// TwinCAT 3 PLC project PLC_SJ_MOCVD
// ProgramVersion: 3.1.4023.0
// libraries:
//   Tc2_ControllerToolbox, * (Beckhoff Automation GmbH)
//   Tc2_IoFunctions, * (Beckhoff Automation GmbH)
//   Tc2_ModbusRTU, * (Beckhoff Automation GmbH)
//   Tc2_ModbusSrv, * (Beckhoff Automation GmbH)
//   Tc2_SerialCom, * (Beckhoff Automation GmbH)
//   Tc2_Standard, * (Beckhoff Automation GmbH)
//   Tc2_System, * (Beckhoff Automation GmbH)
//   Tc2_TempController, * (Beckhoff Automation GmbH)
//   Tc2_Utilities, * (Beckhoff Automation GmbH)
//   Tc3_Module, * (Beckhoff Automation GmbH)
// project tree:
//   GVLs/ GVL_CMD.TcGVL, GVL_IO.TcGVL (not stored), GVL_P2P.TcGVL (not stored), GVL_OP_D.TcGVL (not stored), GVL_COM.TcGVL (not stored), GVL_OP_A.TcGVL (not stored)
//   / PlcTask.TcTTO (not stored), PlcTask_1ms.TcTTO (not stored)
//   POUs/FunctionBlock/ FB_Ramp_0.TcPOU (not stored), FB_RcpRamp.TcPOU, FB_AI_STATUS_Check.TcPOU (not stored), FB_AVG10.TcPOU, FB_DeviationCheck.TcPOU, FB_NoiseCheck.TcPOU (not stored), FB_PID.TcPOU (not stored), FB_Ramp2.TcPOU (not stored), FB_RampControl.TcPOU (not stored)
//   POUs/Function/ F_ET2Sec.TcPOU (not stored), F_LH_PV.TcPOU, F_LH_SV.TcPOU, F_TB_PV2REAL.TcPOU (not stored), F_TB_Rx_BCC.TcPOU (not stored), F_TB_SV2STR.TcPOU (not stored), F_TB_Tx_BCC.TcPOU (not stored), F_Int2Real.TcPOU (not stored), F_OPSTATE.TcPOU (not stored)
//   POUs/ P00_OP.TcPOU (not stored), P01_Init_N_Retain.TcPOU (not stored), P02_Init_MC.TcPOU (not stored), P12_Rx_IH.TcPOU (not stored), P43_SH_UpDw.TcPOU (not stored), P63_Tx_IH.TcPOU (not stored), REF_P02_KL1501.TcPOU (not stored), P15_AI.TcPOU (not stored), P13_DI_N_Check.TcPOU (not stored), P11_Rx_TV.TcPOU (not stored), P22_RCP_Ctrl.TcPOU (not stored), P62_Tx_TV.TcPOU (not stored), P54_DO_ETC.TcPOU (not stored), P31_BypassV.TcPOU (not stored), P21_AL_WN.TcPOU (not stored), P00_Main.TcPOU (not stored), P24_Rot_Calibration.TcPOU (not stored), P25_US_Ctrl.TcPOU (not stored), P61_AO.TcPOU (not stored), P53_DO_VV.TcPOU (not stored), P41_DOR_VAC.TcPOU (not stored), P41_DOR_VAC_Check.TcPOU (not stored), P42_DOR_ATM.TcPOU (not stored), P49_MO_SRC.TcPOU (not stored)
//   POUs/P02_P2P/ P00_Task_Fast.TcPOU (not stored), P2P_LH.TcPOU (not stored), P2P_TB.TcPOU (not stored), Task_Fast_LH.TcPOU (not stored), Task_Fast_TB.TcPOU (not stored), P02_P2P.TcPOU (not stored)
// real-time tasks:
//   TASK PlcTask_Standard: cycle T#10ms, priority 20, ADS port 350
//   TASK PlcTask_Fast: cycle T#2ms, priority 19, ADS port 351
// I/O:
//   DEVICE Device 1 (EtherCAT), AmsNetId 5.62.179.198.2.1
//     Term 1 (EK1200) [EK1200-5000 EtherCAT Power supply (2A E-Bus)]
//       Term 2 (EL6752) [EL6752 DeviceNet Master]
//       Term 3 (EL9011) [EL9011 End Terminal]
//   DEVICE Device 3 (NOV-DP-RAM)
//     Box 6 (Retain Handler)
//   DEVICE Device 2 (EL6752), AmsNetId 5.62.179.198.3.1
//     Box 1  (BK5220) // Bus Coupler
//     Box 2  (BK5220) // Bus Coupler
//     N4E0-T7D2 1 // EDS-File: 'OPP6-2D.EDS' DescText: OPP6-2D Vendor: CKD Corporation Device Type: Generic Device Product Name: OPP6-2D Catalog Number:
//     E3508 // EDS-File: '3500-2.3_SC.EDS' DescText: Eurotherm 3500 Vendor: Eurotherm Device Type: Generic Product Name: Eurotherm 3500 Catalog Number:
//     N4E0-T7D2 2 // EDS-File: 'OPP6-2D.EDS' DescText: OPP6-2D Vendor: CKD Corporation Device Type: Generic Device Product Name: OPP6-2D Catalog Number:
//     Box 10 (IQ-Plus) // EDS-File: 'TBJQPDNG-L041X01 155OUT154.EDS' DescText: Intellisys IQ-Plus Vendor: Nor-Cal Products Device Type: Process Control Valve Product Name: INTELLISYS Catalog Number: IQ-Plus
// variable links:
//   PLC_SJ_MOCVD/PLC_SJ_MOCVD Instance <-> Device 2 (EL6752)
//     PlcTask Inputs/GVL_IO.N_NET_STATES[0] <-> Inputs/Error
//   PLC_SJ_MOCVD/PLC_SJ_MOCVD Instance <-> Device 2 (EL6752)/Box 1  (BK5220)
//     PlcTask Inputs/GVL_IO.N_COUPLER_STATES[0] <-> Inputs/CouplerState
//     PlcTask Inputs/GVL_IO.N_NET_STATES[1] <-> Inputs/MacState
//     PlcTask Inputs/GVL_IO.XA_M01 <-> Term 15 (KL3464)/Channel 1/Data
//     PlcTask Inputs/GVL_IO.XA_M02 <-> Term 15 (KL3464)/Channel 2/Data
//     PlcTask Inputs/GVL_IO.XA_M03 <-> Term 15 (KL3464)/Channel 3/Data
//     PlcTask Inputs/GVL_IO.XA_M04 <-> Term 15 (KL3464)/Channel 4/Data
//     PlcTask Inputs/GVL_IO.XA_M05 <-> Term 17 (KL3464)/Channel 1/Data
//     PlcTask Inputs/GVL_IO.XA_M06 <-> Term 17 (KL3464)/Channel 2/Data
//     PlcTask Inputs/GVL_IO.XA_M07 <-> Term 17 (KL3464)/Channel 3/Data
//     PlcTask Inputs/GVL_IO.XA_M08 <-> Term 17 (KL3464)/Channel 4/Data
//     PlcTask Inputs/GVL_IO.XD_15 <-> Term 3 (KL1408)/Channel 7/Input
//     PlcTask Inputs/GVL_IO.XD_26 <-> Term 5 (KL1408)/Channel 2/Input
//     PlcTask Inputs/GVL_IO.XD_27 <-> Term 5 (KL1408)/Channel 3/Input
//     PlcTask Inputs/GVL_IO.XD_54 <-> Term 8 (KL1408)/Channel 6/Input
//     PlcTask Inputs/GVL_IO.XD_55 <-> Term 8 (KL1408)/Channel 7/Input
//     PlcTask Inputs/GVL_IO.XD_56 <-> Term 8 (KL1408)/Channel 8/Input
//     PlcTask Inputs/GVL_IO.XD_69 <-> Term 10 (KL1408)/Channel 5/Input
//     PlcTask Inputs/GVL_IO.XD_70 <-> Term 10 (KL1408)/Channel 6/Input
//     PlcTask Inputs/GVL_IO.XD_71 <-> Term 10 (KL1408)/Channel 7/Input
//     PlcTask Inputs/GVL_IO.XD_72 <-> Term 10 (KL1408)/Channel 8/Input
//     PlcTask Inputs/GVL_IO.XD_CC_close <-> Term 5 (KL1408)/Channel 1/Input
//     PlcTask Inputs/GVL_IO.XD_CDA_ok <-> Term 3 (KL1408)/Channel 1/Input
//     PlcTask Inputs/GVL_IO.XD_DOR_ATM <-> Term 2 (KL1408)/Channel 6/Input
//     PlcTask Inputs/GVL_IO.XD_DOR_VAC <-> Term 2 (KL1408)/Channel 5/Input
//     PlcTask Inputs/GVL_IO.XD_GC_close <-> Term 4 (KL1408)/Channel 8/Input
//     PlcTask Inputs/GVL_IO.XD_GC_lamp <-> Term 2 (KL1408)/Channel 4/Input
//     PlcTask Inputs/GVL_IO.XD_H2_GC_fail <-> Term 8 (KL1408)/Channel 5/Input
//     PlcTask Inputs/GVL_IO.XD_IH_CB <-> Term 5 (KL1408)/Channel 8/Input
//     PlcTask Inputs/GVL_IO.XD_IH_busy <-> Term 3 (KL1408)/Channel 4/Input
//     PlcTask Inputs/GVL_IO.XD_IH_fail <-> Term 3 (KL1408)/Channel 5/Input
//     PlcTask Inputs/GVL_IO.XD_IH_ready <-> Term 3 (KL1408)/Channel 3/Input
//     PlcTask Inputs/GVL_IO.XD_LAMP_CP <-> Term 6 (KL1408)/Channel 7/Input
//     PlcTask Inputs/GVL_IO.XD_LH{1..8}_CP <-> Term 7 (KL1408)/Channel {1..8}/Input  (8 links)
//     PlcTask Inputs/GVL_IO.XD_LH_CB <-> Term 6 (KL1408)/Channel 3/Input
//     PlcTask Inputs/GVL_IO.XD_LIFT_CP <-> Term 6 (KL1408)/Channel 5/Input
//     PlcTask Inputs/GVL_IO.XD_MAINT <-> Term 2 (KL1408)/Channel 1/Input
//     PlcTask Inputs/GVL_IO.XD_MFC_CP <-> Term 6 (KL1408)/Channel 8/Input
//     PlcTask Inputs/GVL_IO.XD_N2_GC_fail <-> Term 8 (KL1408)/Channel 4/Input
//     PlcTask Inputs/GVL_IO.XD_NH3_GC_fail <-> Term 8 (KL1408)/Channel 2/Input
//     PlcTask Inputs/GVL_IO.XD_PCW_ok <-> Term 3 (KL1408)/Channel 2/Input
//     PlcTask Inputs/GVL_IO.XD_RC_close <-> Term 4 (KL1408)/Channel 7/Input
//     PlcTask Inputs/GVL_IO.XD_RC_lamp <-> Term 2 (KL1408)/Channel 3/Input
//     PlcTask Inputs/GVL_IO.XD_ROT_CP <-> Term 6 (KL1408)/Channel 4/Input
//     PlcTask Inputs/GVL_IO.XD_ROT_fail <-> Term 3 (KL1408)/Channel 6/Input
//     PlcTask Inputs/GVL_IO.XD_RST <-> Term 2 (KL1408)/Channel 2/Input
//     PlcTask Inputs/GVL_IO.XD_SCRUBBER_fail <-> Term 8 (KL1408)/Channel 1/Input
//     PlcTask Inputs/GVL_IO.XD_SH_dw <-> Term 2 (KL1408)/Channel 8/Input
//     PlcTask Inputs/GVL_IO.XD_SH_hi_limit <-> Term 4 (KL1408)/Channel 5/Input
//     PlcTask Inputs/GVL_IO.XD_SH_lo_limit <-> Term 4 (KL1408)/Channel 6/Input
//     PlcTask Inputs/GVL_IO.XD_SH_up <-> Term 2 (KL1408)/Channel 7/Input
//     PlcTask Inputs/GVL_IO.XD_SMPS{1..4}_err <-> Term 5 (KL1408)/Channel {4..7}/Input  (4 links)
//     PlcTask Inputs/GVL_IO.XD_SiH4_GC_fail <-> Term 8 (KL1408)/Channel 3/Input
//     PlcTask Inputs/GVL_IO.XD_TB1_Y_off <-> Term 9 (KL1408)/Channel 2/Input
//     PlcTask Inputs/GVL_IO.XD_TB2_Y_off <-> Term 9 (KL1408)/Channel 4/Input
//     PlcTask Inputs/GVL_IO.XD_TB3_Y_off <-> Term 9 (KL1408)/Channel 6/Input
//     PlcTask Inputs/GVL_IO.XD_TB4_Y_off <-> Term 9 (KL1408)/Channel 8/Input
//     PlcTask Inputs/GVL_IO.XD_TB5_Y_off <-> Term 10 (KL1408)/Channel 2/Input
//     PlcTask Inputs/GVL_IO.XD_TB6_Y_off <-> Term 10 (KL1408)/Channel 4/Input
//     PlcTask Inputs/GVL_IO.XD_TB1_evt <-> Term 9 (KL1408)/Channel 1/Input
//     PlcTask Inputs/GVL_IO.XD_TB2_evt <-> Term 9 (KL1408)/Channel 3/Input
//     PlcTask Inputs/GVL_IO.XD_TB3_evt <-> Term 9 (KL1408)/Channel 5/Input
//     PlcTask Inputs/GVL_IO.XD_TB4_evt <-> Term 9 (KL1408)/Channel 7/Input
//     PlcTask Inputs/GVL_IO.XD_TB5_evt <-> Term 10 (KL1408)/Channel 1/Input
//     PlcTask Inputs/GVL_IO.XD_TB6_evt <-> Term 10 (KL1408)/Channel 3/Input
//     PlcTask Inputs/GVL_IO.XD_TB_CB <-> Term 6 (KL1408)/Channel 1/Input
//     PlcTask Inputs/GVL_IO.XD_TV_CP <-> Term 6 (KL1408)/Channel 6/Input
//     PlcTask Inputs/GVL_IO.XD_VP_CB <-> Term 6 (KL1408)/Channel 2/Input
//     PlcTask Inputs/GVL_IO.XD_VP_al <-> Term 4 (KL1408)/Channel 2/Input
//     PlcTask Inputs/GVL_IO.XD_VP_busy <-> Term 4 (KL1408)/Channel 3/Input
//     PlcTask Inputs/GVL_IO.XD_VP_fail <-> Term 3 (KL1408)/Channel 8/Input
//     PlcTask Inputs/GVL_IO.XD_VP_ready <-> Term 4 (KL1408)/Channel 4/Input
//     PlcTask Inputs/GVL_IO.XD_VP_wn <-> Term 4 (KL1408)/Channel 1/Input
//     PlcTask Outputs/GVL_IO.YA_M01 <-> Term 16 (KL4404)/Channel 1/Data
//     PlcTask Outputs/GVL_IO.YA_M02 <-> Term 16 (KL4404)/Channel 2/Data
//     PlcTask Outputs/GVL_IO.YA_M03 <-> Term 16 (KL4404)/Channel 3/Data
//     PlcTask Outputs/GVL_IO.YA_M04 <-> Term 16 (KL4404)/Channel 4/Data
//     PlcTask Outputs/GVL_IO.YA_M05 <-> Term 18 (KL4404)/Channel 1/Data
//     PlcTask Outputs/GVL_IO.YA_M06 <-> Term 18 (KL4404)/Channel 2/Data
//     PlcTask Outputs/GVL_IO.YA_M07 <-> Term 18 (KL4404)/Channel 3/Data
//     PlcTask Outputs/GVL_IO.YA_M08 <-> Term 18 (KL4404)/Channel 4/Data
//     PlcTask Outputs/GVL_IO.YD_{29..32} <-> Term 14 (KL2408)/Channel {5..8}/Output  (4 links)
//     PlcTask Outputs/GVL_IO.YD_BU <-> Term 11 (KL2408)/Channel 4/Output
//     PlcTask Outputs/GVL_IO.YD_BZ <-> Term 11 (KL2408)/Channel 6/Output
//     PlcTask Outputs/GVL_IO.YD_CC_lamp <-> Term 12 (KL2408)/Channel 8/Output
//     PlcTask Outputs/GVL_IO.YD_DOR_ATM_led <-> Term 14 (KL2408)/Channel 2/Output
//     PlcTask Outputs/GVL_IO.YD_DOR_VAC_led <-> Term 14 (KL2408)/Channel 1/Output
//     PlcTask Outputs/GVL_IO.YD_GC_lamp <-> Term 12 (KL2408)/Channel 7/Output
//     PlcTask Outputs/GVL_IO.YD_GN <-> Term 11 (KL2408)/Channel 3/Output
//     PlcTask Outputs/GVL_IO.YD_IH <-> Term 12 (KL2408)/Channel 1/Output
//     PlcTask Outputs/GVL_IO.YD_IH_mc <-> Term 13 (KL2408)/Channel 1/Output
//     PlcTask Outputs/GVL_IO.YD_IH_rst <-> Term 12 (KL2408)/Channel 2/Output
//     PlcTask Outputs/GVL_IO.YD_LH_mc <-> Term 13 (KL2408)/Channel 4/Output
//     PlcTask Outputs/GVL_IO.YD_RC_lamp <-> Term 12 (KL2408)/Channel 6/Output
//     PlcTask Outputs/GVL_IO.YD_RED <-> Term 11 (KL2408)/Channel 1/Output
//     PlcTask Outputs/GVL_IO.YD_ROT <-> Term 13 (KL2408)/Channel 5/Output
//     PlcTask Outputs/GVL_IO.YD_ROT_break <-> Term 13 (KL2408)/Channel 6/Output
//     PlcTask Outputs/GVL_IO.YD_ROT_rst <-> Term 13 (KL2408)/Channel 7/Output
//     PlcTask Outputs/GVL_IO.YD_RST_led <-> Term 13 (KL2408)/Channel 8/Output
//     PlcTask Outputs/GVL_IO.YD_SH_dw_led <-> Term 14 (KL2408)/Channel 4/Output
//     PlcTask Outputs/GVL_IO.YD_SH_dw_ry <-> Term 11 (KL2408)/Channel 8/Output
//     PlcTask Outputs/GVL_IO.YD_SH_up_led <-> Term 14 (KL2408)/Channel 3/Output
//     PlcTask Outputs/GVL_IO.YD_SH_up_ry <-> Term 11 (KL2408)/Channel 7/Output
//     PlcTask Outputs/GVL_IO.YD_SYS_off_lock <-> Term 12 (KL2408)/Channel 5/Output
//     PlcTask Outputs/GVL_IO.YD_TB_mc <-> Term 13 (KL2408)/Channel 2/Output
//     PlcTask Outputs/GVL_IO.YD_VP <-> Term 12 (KL2408)/Channel 3/Output
//     PlcTask Outputs/GVL_IO.YD_VP_mc <-> Term 13 (KL2408)/Channel 3/Output
//     PlcTask Outputs/GVL_IO.YD_VP_rst <-> Term 12 (KL2408)/Channel 4/Output
//     PlcTask Outputs/GVL_IO.YD_WH <-> Term 11 (KL2408)/Channel 5/Output
//     PlcTask Outputs/GVL_IO.YD_YE <-> Term 11 (KL2408)/Channel 2/Output
//   PLC_SJ_MOCVD/PLC_SJ_MOCVD Instance <-> Device 2 (EL6752)/Box 10 (IQ-Plus)
//     PlcTask Inputs/GVL_P2P.Rx_TV_CDG1_H <-> Connection (Poll)/Inputs/Input 155_5
//     PlcTask Inputs/GVL_P2P.Rx_TV_CDG2_H <-> Connection (Poll)/Inputs/Input 155_3
//     PlcTask Inputs/GVL_P2P.Rx_TV_CDG1_L <-> Connection (Poll)/Inputs/Input 155_4
//     PlcTask Inputs/GVL_P2P.Rx_TV_CDG2_L <-> Connection (Poll)/Inputs/Input 155_2
//     PlcTask Inputs/GVL_P2P.Rx_TV_POS_H <-> Connection (Poll)/Inputs/Input 155_9
//     PlcTask Inputs/GVL_P2P.Rx_TV_POS_L <-> Connection (Poll)/Inputs/Input 155_8
//     PlcTask Inputs/GVL_P2P.Rx_TV_SP_H <-> Connection (Poll)/Inputs/Input 155_7
//     PlcTask Inputs/GVL_P2P.Rx_TV_SP_L <-> Connection (Poll)/Inputs/Input 155_6
//     PlcTask Inputs/GVL_P2P.Rx_TV_ST <-> Connection (Poll)/Inputs/Input 155_1
//     PlcTask Outputs/GVL_P2P.Tx_TV_Arr <-> Connection (Poll)/Outputs/Output 154
//   PLC_SJ_MOCVD/PLC_SJ_MOCVD Instance <-> Device 2 (EL6752)/Box 2  (BK5220)
//     PlcTask Inputs/GVL_IO.N_COUPLER_STATES[1] <-> Inputs/CouplerState
//     PlcTask Inputs/GVL_IO.N_NET_STATES[2] <-> Inputs/MacState
//     PlcTask Inputs/GVL_IO.XA_30 <-> Term 30 (KL3464)/Channel 2/Data
//     PlcTask Inputs/GVL_IO.XA_31 <-> Term 30 (KL3464)/Channel 3/Data
//     PlcTask Inputs/GVL_IO.XA_32 <-> Term 30 (KL3464)/Channel 4/Data
//     PlcTask Inputs/GVL_IO.XA_38 <-> Term 32 (KL3152)/Channel 2/Data
//     PlcTask Inputs/GVL_IO.XA_41 <-> Term 33 (KL3204)/Channel 3/Data
//     PlcTask Inputs/GVL_IO.XA_42 <-> Term 33 (KL3204)/Channel 4/Data
//     PlcTask Inputs/GVL_IO.XA_E01 <-> Term 24 (KL3464)/Channel 4/Data
//     PlcTask Inputs/GVL_IO.XA_E02 <-> Term 26 (KL3464)/Channel 1/Data
//     PlcTask Inputs/GVL_IO.XA_E03 <-> Term 26 (KL3464)/Channel 2/Data
//     PlcTask Inputs/GVL_IO.XA_E04 <-> Term 26 (KL3464)/Channel 3/Data
//     PlcTask Inputs/GVL_IO.XA_E05 <-> Term 26 (KL3464)/Channel 4/Data
//     PlcTask Inputs/GVL_IO.XA_E06 <-> Term 28 (KL3464)/Channel 1/Data
//     PlcTask Inputs/GVL_IO.XA_E07 <-> Term 28 (KL3464)/Channel 2/Data
//     PlcTask Inputs/GVL_IO.XA_IH_CW <-> Term 33 (KL3204)/Channel 2/Data
//     PlcTask Inputs/GVL_IO.XA_M09 <-> Term 20 (KL3464)/Channel 1/Data
//     PlcTask Inputs/GVL_IO.XA_M10 <-> Term 20 (KL3464)/Channel 2/Data
//     PlcTask Inputs/GVL_IO.XA_M11 <-> Term 20 (KL3464)/Channel 3/Data
//     PlcTask Inputs/GVL_IO.XA_M12 <-> Term 20 (KL3464)/Channel 4/Data
//     PlcTask Inputs/GVL_IO.XA_M13 <-> Term 22 (KL3464)/Channel 1/Data
//     PlcTask Inputs/GVL_IO.XA_M14 <-> Term 22 (KL3464)/Channel 2/Data
//     PlcTask Inputs/GVL_IO.XA_M15 <-> Term 22 (KL3464)/Channel 3/Data
//     PlcTask Inputs/GVL_IO.XA_M16 <-> Term 22 (KL3464)/Channel 4/Data
//     PlcTask Inputs/GVL_IO.XA_M17 <-> Term 24 (KL3464)/Channel 1/Data
//     PlcTask Inputs/GVL_IO.XA_M18 <-> Term 24 (KL3464)/Channel 2/Data
//     PlcTask Inputs/GVL_IO.XA_M19 <-> Term 24 (KL3464)/Channel 3/Data
//     PlcTask Inputs/GVL_IO.XA_P02 <-> Term 28 (KL3464)/Channel 3/Data
//     PlcTask Inputs/GVL_IO.XA_P03 <-> Term 28 (KL3464)/Channel 4/Data
//     PlcTask Inputs/GVL_IO.XA_ROT <-> Term 31 (KL3054)/Channel 4/Data
//     PlcTask Inputs/GVL_IO.XA_S01 <-> Term 31 (KL3054)/Channel 1/Data
//     PlcTask Inputs/GVL_IO.XA_S02 <-> Term 31 (KL3054)/Channel 2/Data
//     PlcTask Inputs/GVL_IO.XA_S03 <-> Term 31 (KL3054)/Channel 3/Data
//     PlcTask Inputs/GVL_IO.XA_S04 <-> Term 32 (KL3152)/Channel 1/Data
//     PlcTask Inputs/GVL_IO.XA_S05 <-> Term 30 (KL3464)/Channel 1/Data
//     PlcTask Inputs/GVL_IO.XA_SH_CW <-> Term 33 (KL3204)/Channel 1/Data
//     PlcTask Outputs/GVL_IO.YA_E01 <-> Term 25 (KL4404)/Channel 4/Data
//     PlcTask Outputs/GVL_IO.YA_E02 <-> Term 27 (KL4404)/Channel 1/Data
//     PlcTask Outputs/GVL_IO.YA_E03 <-> Term 27 (KL4404)/Channel 2/Data
//     PlcTask Outputs/GVL_IO.YA_E04 <-> Term 27 (KL4404)/Channel 3/Data
//     PlcTask Outputs/GVL_IO.YA_E05 <-> Term 27 (KL4404)/Channel 4/Data
//     PlcTask Outputs/GVL_IO.YA_E06 <-> Term 29 (KL4404)/Channel 1/Data
//     PlcTask Outputs/GVL_IO.YA_E07 <-> Term 29 (KL4404)/Channel 2/Data
//     PlcTask Outputs/GVL_IO.YA_M09 <-> Term 21 (KL4404)/Channel 1/Data
//     PlcTask Outputs/GVL_IO.YA_M10 <-> Term 21 (KL4404)/Channel 2/Data
//     PlcTask Outputs/GVL_IO.YA_M11 <-> Term 21 (KL4404)/Channel 3/Data
//     PlcTask Outputs/GVL_IO.YA_M12 <-> Term 21 (KL4404)/Channel 4/Data
//     PlcTask Outputs/GVL_IO.YA_M13 <-> Term 23 (KL4404)/Channel 1/Data
//     PlcTask Outputs/GVL_IO.YA_M14 <-> Term 23 (KL4404)/Channel 2/Data
//     PlcTask Outputs/GVL_IO.YA_M15 <-> Term 23 (KL4404)/Channel 3/Data
//     PlcTask Outputs/GVL_IO.YA_M16 <-> Term 23 (KL4404)/Channel 4/Data
//     PlcTask Outputs/GVL_IO.YA_M17 <-> Term 25 (KL4404)/Channel 1/Data
//     PlcTask Outputs/GVL_IO.YA_M18 <-> Term 25 (KL4404)/Channel 2/Data
//     PlcTask Outputs/GVL_IO.YA_M19 <-> Term 25 (KL4404)/Channel 3/Data
//     PlcTask Outputs/GVL_IO.YA_P03 <-> Term 29 (KL4404)/Channel 3/Data
//     PlcTask Outputs/GVL_IO.YA_ROT <-> Term 29 (KL4404)/Channel 4/Data
//     PlcTask_1ms Inputs/GVL_P2P.in22B_LH/D[{0..21}] <-> Term 34 (KL6031)/Channel 1/Data In {0..21}  (22 links)
//     PlcTask_1ms Inputs/GVL_P2P.in22B_LH/Status <-> Term 34 (KL6031)/Channel 1/State
//     PlcTask_1ms Inputs/GVL_P2P.in22B_TB/D[{0..21}] <-> Term 35 (KL6031)/Channel 1/Data In {0..21}  (22 links)
//     PlcTask_1ms Inputs/GVL_P2P.in22B_TB/Status <-> Term 35 (KL6031)/Channel 1/State
//     PlcTask_1ms Outputs/GVL_P2P.out22B_LH/Ctrl <-> Term 34 (KL6031)/Channel 1/Ctrl
//     PlcTask_1ms Outputs/GVL_P2P.out22B_LH/D[{0..21}] <-> Term 34 (KL6031)/Channel 1/Data Out {0..21}  (22 links)
//     PlcTask_1ms Outputs/GVL_P2P.out22B_TB/Ctrl <-> Term 35 (KL6031)/Channel 1/Ctrl
//     PlcTask_1ms Outputs/GVL_P2P.out22B_TB/D[{0..21}] <-> Term 35 (KL6031)/Channel 1/Data Out {0..21}  (22 links)
//   PLC_SJ_MOCVD/PLC_SJ_MOCVD Instance <-> Device 2 (EL6752)/E3508
//     PlcTask Inputs/GVL_IO.N_NET_STATES[6] <-> Inputs/MacState
//     PlcTask Inputs/GVL_P2P.Rx_IH_AL_H <-> Connection (Poll)/Inputs/Input Data_10
//     PlcTask Inputs/GVL_P2P.Rx_IH_AL_L <-> Connection (Poll)/Inputs/Input Data_9
//     PlcTask Inputs/GVL_P2P.Rx_IH_AM_H <-> Connection (Poll)/Inputs/Input Data_12
//     PlcTask Inputs/GVL_P2P.Rx_IH_AM_L <-> Connection (Poll)/Inputs/Input Data_11
//     PlcTask Inputs/GVL_P2P.Rx_IH_AT_ST_H <-> Connection (Poll)/Inputs/Input Data_14
//     PlcTask Inputs/GVL_P2P.Rx_IH_AT_ST_L <-> Connection (Poll)/Inputs/Input Data_13
//     PlcTask Inputs/GVL_P2P.Rx_IH_D_H <-> Connection (Poll)/Inputs/Input Data_20
//     PlcTask Inputs/GVL_P2P.Rx_IH_D_L <-> Connection (Poll)/Inputs/Input Data_19
//     PlcTask Inputs/GVL_P2P.Rx_IH_I_H <-> Connection (Poll)/Inputs/Input Data_18
//     PlcTask Inputs/GVL_P2P.Rx_IH_I_L <-> Connection (Poll)/Inputs/Input Data_17
//     PlcTask Inputs/GVL_P2P.Rx_IH_MOUT_H <-> Connection (Poll)/Inputs/Input Data_8
//     PlcTask Inputs/GVL_P2P.Rx_IH_MOUT_L <-> Connection (Poll)/Inputs/Input Data_7
//     PlcTask Inputs/GVL_P2P.Rx_IH_PV_H <-> Connection (Poll)/Inputs/Input Data_2
//     PlcTask Inputs/GVL_P2P.Rx_IH_PV_L <-> Connection (Poll)/Inputs/Input Data_1
//     PlcTask Inputs/GVL_P2P.Rx_IH_P_H <-> Connection (Poll)/Inputs/Input Data_16
//     PlcTask Inputs/GVL_P2P.Rx_IH_P_L <-> Connection (Poll)/Inputs/Input Data_15
//     PlcTask Inputs/GVL_P2P.Rx_IH_SV_H <-> Connection (Poll)/Inputs/Input Data_4
//     PlcTask Inputs/GVL_P2P.Rx_IH_SV_L <-> Connection (Poll)/Inputs/Input Data_3
//     PlcTask Inputs/GVL_P2P.Rx_IH_TSV_H <-> Connection (Poll)/Inputs/Input Data_6
//     PlcTask Inputs/GVL_P2P.Rx_IH_TSV_L <-> Connection (Poll)/Inputs/Input Data_5
//     PlcTask Outputs/GVL_P2P.Tx_IH_ABS_HI_H <-> Connection (Poll)/Outputs/Output Data_12
//     PlcTask Outputs/GVL_P2P.Tx_IH_ABS_HI_L <-> Connection (Poll)/Outputs/Output Data_11
//     PlcTask Outputs/GVL_P2P.Tx_IH_AL_CR_H <-> Connection (Poll)/Outputs/Output Data_8
//     PlcTask Outputs/GVL_P2P.Tx_IH_AL_CR_L <-> Connection (Poll)/Outputs/Output Data_7
//     PlcTask Outputs/GVL_P2P.Tx_IH_AM_H <-> Connection (Poll)/Outputs/Output Data_4
//     PlcTask Outputs/GVL_P2P.Tx_IH_AM_L <-> Connection (Poll)/Outputs/Output Data_3
//     PlcTask Outputs/GVL_P2P.Tx_IH_AT_EN_H <-> Connection (Poll)/Outputs/Output Data_10
//     PlcTask Outputs/GVL_P2P.Tx_IH_AT_EN_L <-> Connection (Poll)/Outputs/Output Data_9
//     PlcTask Outputs/GVL_P2P.Tx_IH_MOUT_H <-> Connection (Poll)/Outputs/Output Data_6
//     PlcTask Outputs/GVL_P2P.Tx_IH_MOUT_L <-> Connection (Poll)/Outputs/Output Data_5
//     PlcTask Outputs/GVL_P2P.Tx_IH_TSV_H <-> Connection (Poll)/Outputs/Output Data_2
//     PlcTask Outputs/GVL_P2P.Tx_IH_TSV_L <-> Connection (Poll)/Outputs/Output Data_1
//   PLC_SJ_MOCVD/PLC_SJ_MOCVD Instance <-> Device 2 (EL6752)/N4E0-T7D2 1
//     PlcTask Inputs/GVL_IO.N_NET_STATES[3] <-> Inputs/MacState
//     PlcTask Outputs/GVL_P2P.Tx_SOL1 <-> Connection (Poll)/Outputs/Output Data
//   PLC_SJ_MOCVD/PLC_SJ_MOCVD Instance <-> Device 2 (EL6752)/N4E0-T7D2 2
//     PlcTask Outputs/GVL_P2P.Tx_SOL2 <-> Connection (Poll)/Outputs/Output Data
//   PLC_SJ_MOCVD/PLC_SJ_MOCVD Instance <-> Device 3 (NOV-DP-RAM)/Box 6 (Retain Handler)
//     PlcTask Retains/P01_Init_N_Retain.R_A_SV_AL <-> Retains/P01_Init_N_Retain.R_A_SV_AL_[851]
//     PlcTask Retains/P01_Init_N_Retain.R_A_SV_WN <-> Retains/P01_Init_N_Retain.R_A_SV_WN_[851]
//     PlcTask Retains/P01_Init_N_Retain.R_DevTM_AL <-> Retains/P01_Init_N_Retain.R_DevTM_AL_[851]
//     PlcTask Retains/P01_Init_N_Retain.R_DevTM_WN <-> Retains/P01_Init_N_Retain.R_DevTM_WN_[851]
//     PlcTask Retains/P01_Init_N_Retain.R_Dev_AL <-> Retains/P01_Init_N_Retain.R_Dev_AL_[851]
//     PlcTask Retains/P01_Init_N_Retain.R_Dev_WN <-> Retains/P01_Init_N_Retain.R_Dev_WN_[851]
//     PlcTask Retains/P01_Init_N_Retain.R_EN_AL <-> Retains/P01_Init_N_Retain.R_EN_AL_[851]
//     PlcTask Retains/P01_Init_N_Retain.R_EN_RAMP <-> Retains/P01_Init_N_Retain.R_EN_RAMP_[851]
//     PlcTask Retains/P01_Init_N_Retain.R_EN_RCP_RAMP <-> Retains/P01_Init_N_Retain.R_EN_RCP_RAMP_[851]
//     PlcTask Retains/P01_Init_N_Retain.R_EN_WN <-> Retains/P01_Init_N_Retain.R_EN_WN_[851]
//     PlcTask Retains/P01_Init_N_Retain.R_ETC_A <-> Retains/P01_Init_N_Retain.R_ETC_A_[851]
//     PlcTask Retains/P01_Init_N_Retain.R_ETC_D <-> Retains/P01_Init_N_Retain.R_ETC_D_[851]
//     PlcTask Retains/P01_Init_N_Retain.R_LH_TB_SV <-> Retains/P01_Init_N_Retain.R_LH_TB_SV_[851]
//     PlcTask Retains/P01_Init_N_Retain.R_MAX <-> Retains/P01_Init_N_Retain.R_MAX_[851]
//     PlcTask Retains/P01_Init_N_Retain.R_MIN <-> Retains/P01_Init_N_Retain.R_MIN_[851]
//     PlcTask Retains/P01_Init_N_Retain.R_MS_SET <-> Retains/P01_Init_N_Retain.R_MS_SET_[851]
//     PlcTask Retains/P01_Init_N_Retain.R_PV_ROT_1TURN_PLS <-> Retains/P01_Init_N_Retain.R_PV_ROT_1TURN_PLS_[851]
//     PlcTask Retains/P01_Init_N_Retain.R_PV_ROT_INCH_PLS <-> Retains/P01_Init_N_Retain.R_PV_ROT_INCH_PLS_[851]
//     PlcTask Retains/P01_Init_N_Retain.R_SOL_IDX1 <-> Retains/P01_Init_N_Retain.R_SOL_IDX1_[851]
//     PlcTask Retains/P01_Init_N_Retain.R_SOL_IDX2 <-> Retains/P01_Init_N_Retain.R_SOL_IDX2_[851]
//     PlcTask Retains/P01_Init_N_Retain.R_TV_posMode <-> Retains/P01_Init_N_Retain.R_TV_posMode_[851]
//     PlcTask Retains/P01_Init_N_Retain.R_US_A <-> Retains/P01_Init_N_Retain.R_US_A_[851]
//     PlcTask Retains/P01_Init_N_Retain.R_US_A_EN <-> Retains/P01_Init_N_Retain.R_US_A_EN_[851]
//     PlcTask Retains/P01_Init_N_Retain.R_US_D <-> Retains/P01_Init_N_Retain.R_US_D_[851]

// ---- GVLs/GVL_CMD.TcGVL
//{attribute 'qualified_only'}
VAR_GLOBAL

//Address Test
//B_B1 AT%MX127999.7: BOOL;	
//B_B2 AT%MB127999: BYTE;	
//B_B3 AT%MW63999: WORD;
//B_B4 AT%QW63999: WORD;			
//N_1	AT%MW29600: REAL;
	
//Excel GVL_CMD
cm_TCAT_restart : BOOL;
cm_RST : BOOL;
cm_FC_stop : BOOL;
cm_DOR_VAC : BOOL;
cm_DOR_ATM : BOOL;
cm_RCP_start : BOOL;
cm_ROT_caliStart : BOOL;



cm_RCP_pause : BOOL;
cm_RCP_restart : BOOL;
cm_RCP_skip : BOOL;
cm_RCP_end : BOOL;
cm_RCP_1step : BOOL;
cm_RCP_safeStop : BOOL;
cm_DO_TEST : BOOL;
cm_MAX_save : BOOL;
cm_US_save : BOOL;
cm_AL_save : BOOL;
cm_WN_save : BOOL;
cm_ETC_save : BOOL;
cm_EN_RAMP_save : BOOL;
cm_MO_save : BOOL;
cm_SOL1_save : BOOL;
cm_SOL2_save : BOOL;
cm_US1 : BOOL;
cm_US2 : BOOL;
cm_US3 : BOOL;
cm_US4 : BOOL;
cm_TV_open : BOOL;
cm_TV_close : BOOL;
cm_TV_run : BOOL;
cm_TV_stop : BOOL;
cm_TV_presMode : BOOL;
cm_TV_posMode : BOOL;
cm_ROT_jog : BOOL;
cm_ROT_inch : BOOL;
cm_ROT_pulseZero : BOOL;
cm_BZ_UserStop : BOOL;

cm_MAINT : BOOL;
cm_DEBUG : BOOL;
cm_IHT_AT : BOOL;

cm_MAINT_off : BOOL;
cm_V01 : BOOL;
cm_V02 : BOOL;
cm_V03 : BOOL;
cm_V04 : BOOL;
cm_V05 : BOOL;
cm_V06 : BOOL;
cm_V07 : BOOL;
cm_V08 : BOOL;
cm_V09 : BOOL;
cm_V10 : BOOL;
cm_V11 : BOOL;
cm_V12 : BOOL;
cm_V13 : BOOL;
cm_V14 : BOOL;
cm_V15 : BOOL;
cm_V16 : BOOL;
cm_V17 : BOOL;
cm_V18 : BOOL;
cm_V19 : BOOL;
cm_V20 : BOOL;
cm_V21 : BOOL;
cm_V22 : BOOL;
cm_V23 : BOOL;
cm_V24 : BOOL;
cm_V25 : BOOL;
cm_V26 : BOOL;
cm_V27 : BOOL;
cm_V28 : BOOL;
cm_V29 : BOOL;
cm_V30 : BOOL;
cm_V31 : BOOL;
cm_V32 : BOOL;
cm_V33_1 : BOOL;
cm_V33_2 : BOOL;
cm_V34 : BOOL;
cm_V35 : BOOL;
cm_V36 : BOOL;
cm_V37 : BOOL;
cm_V38 : BOOL;
cm_V39 : BOOL;
cm_V40 : BOOL;
cm_V41 : BOOL;
cm_V42 : BOOL;
cm_V43 : BOOL;
cm_V44 : BOOL;
cm_V45 : BOOL;
cm_V46 : BOOL;
cm_V47 : BOOL;
cm_V48 : BOOL;
cm_V49 : BOOL;
cm_V50 : BOOL;
cm_V51 : BOOL;
cm_V52 : BOOL;

cm_RED : BOOL;
cm_YE : BOOL;
cm_GN : BOOL;
cm_BU : BOOL;
cm_WH : BOOL;
cm_BZ : BOOL;
cm_SH_up_ry : BOOL;
cm_SH_dw_ry : BOOL;
cm_IH : BOOL;
cm_IH_rst : BOOL;
cm_VP : BOOL;
cm_VP_rst : BOOL;
cm_SYS_off_lock : BOOL;
cm_RC_lamp : BOOL;
cm_GC_lamp : BOOL;
cm_CC_lamp : BOOL;
cm_IH_mc : BOOL;
cm_TB_mc : BOOL;
cm_VP_mc : BOOL;
cm_LH_mc : BOOL;
cm_ROT : BOOL;
cm_ROT_break : BOOL;
cm_ROT_rst : BOOL;
cm_RST_led : BOOL;
cm_DOR_VAC_led : BOOL;
cm_DOR_ATM_led : BOOL;
cm_SH_up_led : BOOL;
cm_SH_dw_led : BOOL;
cm_Y_29 : BOOL;
cm_Y_30 : BOOL;
cm_Y_31 : BOOL;
cm_Y_32 : BOOL;


cm_LH1_at : BOOL;
cm_LH2_at : BOOL;
cm_LH3_at : BOOL;
cm_LH4_at : BOOL;
cm_LH5_at : BOOL;
cm_LH6_at : BOOL;
cm_LH7_at : BOOL;
cm_LH8_at : BOOL;


END_VAR

// ---- POUs/FunctionBlock/FB_RcpRamp.TcPOU
FUNCTION_BLOCK FB_RcpRamp
VAR_INPUT
	pEN: BOOL;
	bPause: BOOL;	
	bStop: BOOL;
	fSV: REAL;	
	fSV_Step: REAL;
END_VAR
VAR_OUTPUT
	fyOut: REAL;
END_VAR
VAR_IN_OUT	
END_VAR
VAR
	fSV_Old: REAL;
	fSV_Step_Old: REAL;
	fSV_Inc: REAL;
	isPlus: BOOL;
END_VAR


//Check Input Value changed
IF fSV <> fSV_Old OR fSV_Step <> fSV_Step_Old THEN
	IF fSV_Step	<= 0 THEN 
		fSV_Step := 1; 
	END_IF	
    isPlus := fSV > fyOut;// Check Inc OR Dec
	fSV_Inc := (fyOut - fSV) / fSV_Step; //Calc Inc Value   
END_IF

fSV_Old := fSV;
fSV_Step_Old := fSV_Step;

//Ramping
IF pEN THEN
	IF bPause = 0 THEN
		fyOut := fyOut - fSV_Inc;
	END_IF
		
	IF isPlus = 0 AND fyOut < fSV THEN fyOut := fSV; END_IF
	IF isPlus = 1 AND fyOut > fSV THEN fyOut := fSV; END_IF
END_IF


IF fSV_Step = 1 THEN
	fyOut := fSV;
END_IF

IF bStop THEN
	fSV_Step := 1;
	fSV := fyOut;
END_IF


//T1(IN:=bT1_On, PT:=tTimeUnit);

END_FUNCTION_BLOCK

// ---- POUs/Function/F_LH_PV.TcPOU
FUNCTION F_LH_PV : REAL
VAR_INPUT
	hexPV: STRING;
	nDecimal: INT := 0;
END_VAR
VAR
	data: ARRAY[0..1] OF BYTE;
	b1: BYTE;
	cbData: UDINT;
	ptPV: POINTER TO INT;
	iPV: INT;
	i: INT;
	r1: REAL;
END_VAR


cbData := HEXSTR_TO_DATA(hexPV, ADR(data), SIZEOF(data));
		
//Swap
b1 := data[0];
data[0] := data[1];
data[1] := b1;
		
ptPV := ADR(data);
iPV := ptPV^;
r1 := INT_TO_REAL(iPV);

//Decimal
FOR i := 0 TO nDecimal - 1 BY 1 DO
	r1 := r1 / 10;
END_FOR

F_LH_PV := r1;

END_FUNCTION

// ---- POUs/Function/F_LH_SV.TcPOU
FUNCTION F_LH_SV : STRING
VAR_INPUT
	SV: REAL;
	nDecimal: INT := 0;
END_VAR
VAR
	iPV: INT;
	wPV: WORD;
	i: INT;
	r1: REAL;
END_VAR


r1 := SV;

//Decimal
FOR i := 0 TO nDecimal - 1 BY 1 DO
	r1 := r1 * 10;
END_FOR

iPV := REAL_TO_INT(r1);
wPV := INT_TO_WORD(iPV);

F_LH_SV := WORD_TO_HEXSTR(in:= wPV, iPrecision:= 4, bLoCase:= FALSE);

END_FUNCTION

// ---- POUs/FunctionBlock/FB_AVG10.TcPOU
FUNCTION_BLOCK FB_AVG10
VAR_INPUT
	fValue: REAL;
END_VAR
VAR_OUTPUT
	AVG: REAL := 0;
END_VAR
VAR
	Datas: ARRAY [0..9] OF REAL;
	Total: REAL := 0;	
    i: INT := 0;
	j: INT := 0;
END_VAR


IF i = 9 THEN
	//First In -> First Out
	FOR j := 1 TO 9 DO
		Datas[j-1] := Datas[j];
	END_FOR 
	Datas[9] := fValue;
ELSE
	Datas[i] := fValue;
	i := i + 1;
END_IF

Total := 0;
FOR j := 0 TO 9 DO
	Total := Total + Datas[j];
END_FOR 

AVG := Total / 10;

END_FUNCTION_BLOCK

// ---- POUs/FunctionBlock/FB_DeviationCheck.TcPOU
FUNCTION_BLOCK FB_DeviationCheck
VAR_INPUT
	bReset: BOOL;
	bEn_Alarm: BOOL;
	bEn_Warning: BOOL;
	fDeviPV: REAL;
	wAlarmDevi: WORD;
	dwAlarmCheckMilisec: DWORD;
	wWarningDevi: WORD;
	dwWarningCheckMilisec: DWORD;	
END_VAR
VAR_OUTPUT
	isAlarm : BOOL;
	isWarning : BOOL;
END_VAR
VAR
	T1 : TON;
	T2 : TON;
	wAlarmDev_Old : WORD;
	wWarnDev_Old : WORD;
	fAlarmDev : REAL;
	fWarnDev : REAL;
END_VAR

//Alarm Check
IF wAlarmDevi <> wAlarmDev_Old THEN
	wAlarmDev_Old := wAlarmDevi;
	fAlarmDev := WORD_TO_REAL(wAlarmDev_Old);
END_IF

T1();
T1.PT := DWORD_TO_TIME(dwAlarmCheckMilisec);
T1.IN := bEn_Alarm AND ABS(fDeviPV) > fAlarmDev AND isAlarm = FALSE ;
IF T1.Q THEN
	isAlarm := TRUE;
END_IF;


//Warning Check
IF wWarningDevi <> wWarnDev_Old THEN
	wWarnDev_Old := wWarningDevi;
	fWarnDev := WORD_TO_REAL(wWarnDev_Old);
END_IF

T2();
T2.PT := DWORD_TO_TIME(dwWarningCheckMilisec);
T2.IN := bEn_Warning AND ABS(fDeviPV) > fWarnDev AND isWarning = FALSE ;
IF T2.Q THEN
	isWarning := TRUE;
END_IF;

IF bReset THEN
	isAlarm := FALSE;	
	isWarning := FALSE;
END_IF

END_FUNCTION_BLOCK
